PROGRAM MAIN
VAR
END_VAR

//Apparatskåp
AS101();
KV1();
S1();
VVC1();

END_PROGRAM

(* stored: Version 1.1.0.1, ProductVersion 3.1.4024.13
   POU MAIN: Id {a2945148-3502-4861-8d96-4b8191e12331}, SpecialFunc None *)
